# EPICS substitutions: db/Beckhoff_1XXX/ecmcEK1122.substitutions
file ecmcEcSlave.template
{
  pattern {}
          {}
}
